// TIA Portal V21 export
DATA_BLOCK "CicloScansioneCPU_I"   // DB8
AUTHOR : Roman
FAMILY : BrainElectric
NAME : 89
VERSION : 1.3
// stored: AutoNumber false, InstanceOfName CicloScansioneCPU_G, InstanceOfType FB
"CicloScansioneCPU_G"
   // VAR_INPUT
   //    I_PrimoCicloCpu : Bool := FALSE;
   // END_VAR
   // VAR
   //    l_lrCicloCpu { ExternalAccessible := 'False'; ExternalVisible := 'False'; ExternalWritable := 'False'} : LReal := 0.0743422844444444;
   //    l_lrCicloCpuMem { ExternalAccessible := 'False'; ExternalVisible := 'False'; ExternalWritable := 'False'} : LReal := 16#0003_2FC2_DE58_DEF6;
   //    l_rCicloCpuResto : LReal := 0.205517246914266;
   //    O_rCicloCpu : Real := 0.07434229;
   //    O_iCicloCpu : Int := 74;
   // END_VAR
BEGIN
END_DATA_BLOCK
